Staubli VAL3: dateBase.dtx

public bool bCenterPoint = true
public bool bFrameTeach = true
public bool bPLC
public bool bToolTeach
public bool bWorTbMoving
public frame fWorkTable = {x=1460.596362, y=35.712914, z=-199.189903, rx=-0.117127, ry=-0.30554, rz=-53.750077, fatherId=world[0]}
public jointRx jHome = {j1=11.40774, j2=30.671658, j3=109.333141, j4=204.624689, j5=51.130912, j6=-196.428273}
public mdesc mGrindingSpd = {accel=70, decel=70, tmax=100, leave=0.5, reach=0.5}
public mdesc mNomSpeed = {accel=36, vel=60, decel=36, rmax=2000, tmax=100, blend=cartesian, leave=5, reach=5}
public num nPrdRadius = 100.111913
public tool tTCP = {x=1.417, y=48.029, z=261.326, rx=-28.407, ry=-42.029, rz=-19.448, fatherId=flange[0], ioLink=valve1}
